Staubli VAL3: setAxis.pgx

public program setAxis(num x_nAxisNum)
begin
  switch x_nAxisNum
    case 6
      nAxisNum=6
    break
    case 4
      nAxisNum=4
    break
    default
      popUpMsg("请输入正确的关节数目!")
    break
  endSwitch
end
